// TIA Portal project "Semaforo" (V15)
// Ejemplo con fines didacticos

(* hardware
DEVICE "HMI_1"  KTP700 Basic PN
   slot 0: "HMI_1"  KTP700 Basic PN  6AV2 123-2GB03-0AX0  15.0.0.0
   slot 1: "HMI_RT_1"  KTP700 Basic PN  6AV2 123-2GB03-0AX0  15.0.0.0
   slot 5: "HMI_1.IE_CP_1"  PROFINET Interface  15.0.0.0
      slot 1: "Interfaz PROFINET_1"  PROFINET Interface
         slot 1: "Port_1"  Port
DEVICE "S7-1200 station_1"  S7-1200 Station
   slot 0: "Rack_0"  S7-1200 Rack  Rack  V1.0
   slot 1: "PLC_1"  CPU 1212C DC/DC/DC  6ES7 212-1AE40-0XB0  V4.2
*)

// ===== PLC "PLC_1"  CPU 1212C DC/DC/DC =====

VAR_GLOBAL   // PLC tag table "Tabla de variables estándar"
   "marcha" AT %M0.0 : Bool;   // Marcha
   "verde" AT %Q0.0 : Bool;   // Luz verde
END_VAR

// folder: System blocks/Program resources

DATA_BLOCK "temporizadoVerde"   // DB1
{ S7_Optimized_Access := 'TRUE' }
AUTHOR : Simatic
FAMILY : IEC
NAME : IEC_TMR
VERSION : 1.0
// stored: InstanceOfName IEC_TIMER
"IEC_TIMER"
BEGIN
END_DATA_BLOCK

// folder: (top level)

ORGANIZATION_BLOCK "Main"   // OB1, LAD, ProgramCycle
TITLE = "Main Program Sweep (Cycle)"
{ S7_Optimized_Access := 'TRUE' }
VERSION : 0.1
   VAR_INPUT
      Initial_Call : Bool;   // Initial call of this OB
      Remanence : Bool;   // =True, if remanent data are available
   END_VAR
BEGIN

REGION Network 1: Luz verde
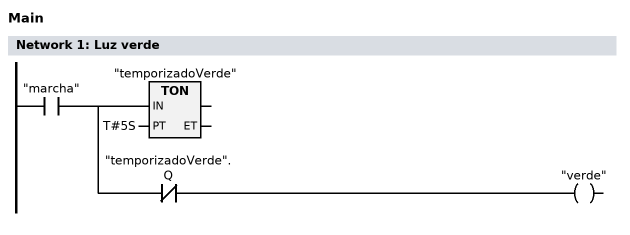
   "temporizadoVerde".TON(IN := "marcha", PT := T#5S);
   "verde" := "marcha" AND NOT "temporizadoVerde".Q;
END_REGION
END_ORGANIZATION_BLOCK

(* ===== HMI "HMI_RT_1" =====
system functions are stored by id; their names below are inferred from use
connection "HMI_Conexión_1": ETHERNET, SMART_S7_1200_OMS

HMI tags "Tabla de variables estándar"
   "Número_imagen_variable" : UInt, internal
   "marcha" : Bool = PLC marcha AT %M0.0, 1 s

text list "Nombre_imagen_lista_texto": 1 'Imagen raíz'

Template "Plantilla_1" 800x480
   DateTimeField "HmiScreenItemData" at 695,25 size 105x25
   DateTimeField "HmiScreenItemData_1" at 695,0 size 105x25
   GraphicView "Plantilla_Visor de gráficos_1" at 5,4 size 120x77; Picture "pelota"
   GraphicView "Plantilla_Visor de gráficos_2" at 244,146 size 281x310; Picture "semaforo01_2"
   Button "Plantilla_Botón_1" at 239,83 size 129x42; TextOff 'MARCHA'
      on Press: SetBit("marcha")
   Button "Plantilla_Botón_2" at 410,85 size 138x42; TextOn 'PARADA'; TextOff 'PARADA'
      on Press: ResetBit("marcha")

screen "Imagen raíz" 800x480, template "Plantilla_1"
   on GenerateScreen: SetTag("Número_imagen_variable", 1)
*)